FUNCTION_BLOCK ConveyorCTLMultiCast (* Basic Function Block Type *)
  (* Standard: 61499-2 *)
  (* Version 0.2, 2003-12-04, JHC, Rockwell Automation, Renamed for better indexing. *)
  (* Version 0.1, 2002-11-05, JHC, Rockwell Automation, Corrected missing ST element in Algorithm REQ. *)
  (* Version 0.0, 2000-05-30, JHC, Rockwell Automation *)
  (* Compiler header: package fb.rt.cs725; *)
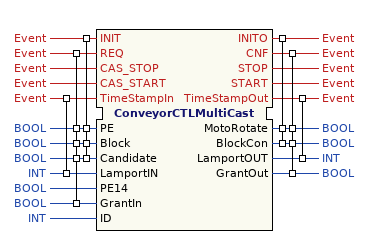
  EVENT_INPUT
    INIT WITH PE, Block, Candidate; (* Initialization Request *)
    REQ WITH PE, Block, Candidate, GrantIn; (* Normal Execution Request *)
    CAS_STOP;
    CAS_START;
    TimeStampIn WITH LamportIN;
  END_EVENT
  EVENT_OUTPUT
    INITO WITH MotoRotate, BlockCon; (* Initialization Confirm *)
    CNF WITH MotoRotate, BlockCon, GrantOut; (* Execution Confirmation *)
    STOP;
    START;
    TimeStampOut WITH LamportOUT;
  END_EVENT
  VAR_INPUT
    PE : BOOL; (* Input event qualifier *)
    Block : BOOL;
    Candidate : BOOL;
    LamportIN : INT;
    PE14 : BOOL;
    GrantIn : BOOL;
    ID : INT;
  END_VAR
  VAR_OUTPUT
    MotoRotate : BOOL; (* Output event qualifier *)
    BlockCon : BOOL;
    LamportOUT : INT;
    GrantOut : BOOL;
  END_VAR
  VAR
    lastPE : BOOL := 1;
    lastBlock : BOOL := 0;
    lamportClock : INT;
  END_VAR
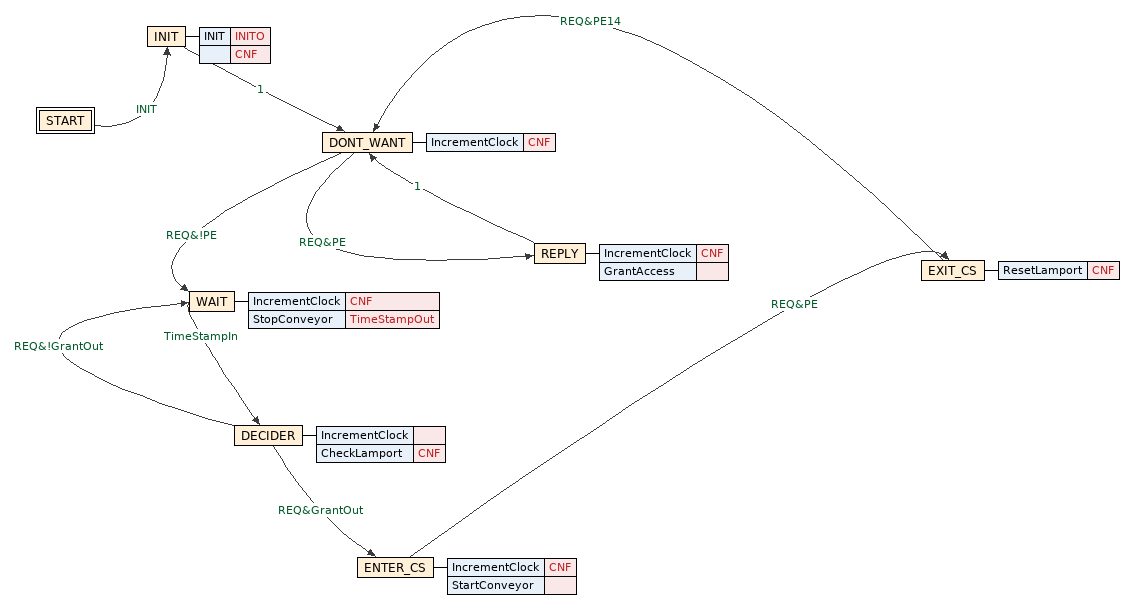
  EC_STATES
    START; (* Initial State *)
    INIT : INIT -> INITO, -> CNF; (* Initialization *)
    WAIT : IncrementClock -> CNF, StopConveyor -> TimeStampOut;
    DONT_WANT : IncrementClock -> CNF;
    REPLY : IncrementClock -> CNF, GrantAccess;
    DECIDER : IncrementClock, CheckLamport -> CNF;
    ENTER_CS : IncrementClock -> CNF, StartConveyor;
    EXIT_CS : ResetLamport -> CNF;
  END_STATES
  EC_TRANSITIONS
    START TO INIT := INIT;
    INIT TO DONT_WANT := 1;
    DONT_WANT TO WAIT := REQ&!PE;
    DONT_WANT TO REPLY := REQ&PE;
    REPLY TO DONT_WANT := 1;
    WAIT TO DECIDER := TimeStampIn;
    DECIDER TO WAIT := REQ&!GrantOut;
    DECIDER TO ENTER_CS := REQ&GrantOut;
    ENTER_CS TO EXIT_CS := REQ&PE;
    EXIT_CS TO DONT_WANT := REQ&PE14;
  END_TRANSITIONS
  ALGORITHM INIT IN ST: (* Initialization algorithm *)
MotoRotate := TRUE;
Block := FALSE;
lamportClock := 0;
GrantOut := FALSE;

System.out.println(this + " " + MotoRotate);
System.out.println(MotoRotate);
  END_ALGORITHM
  ALGORITHM REQ IN ST: (* Normally executed algorithm *)
System.out.println(this +  " -> Candidate" + Candidate);
IF Candidate THEN
IF lastPE !:= PE THEN
IF NOT PE THEN
BlockCon:= TRUE;
System.out.println("BlockCon = true");
ELSE
BlockCon:=FALSE;
System.out.println("BlockCon = false");
END_IF
lastPE := PE;
END_IF
IF lastBlock !:= Block THEN
IF Block THEN
STOP.serviceEvent(this);
MotoRotate := FALSE;
System.out.println("Cas Stop");
ELSE
START.serviceEvent(this);
MotoRotate := TRUE;
System.out.println("Cas Start");
END_IF
lastBlock := Block;
END_IF
END_IF
  END_ALGORITHM
  ALGORITHM START IN ST:
MotoRotate:=TRUE;
System.out.println(this + " Start " + MotoRotate);

System.out.println("Start " + MotoRotate);
  END_ALGORITHM
  ALGORITHM STOP IN ST:
MotoRotate := FALSE;
System.out.println(this + " Stop " + MotoRotate);

System.out.println("Stop " + MotoRotate);
  END_ALGORITHM
  ALGORITHM CheckLamport IN Java:
if(LamportIN.value < lamportClock.value){
GrantOut.value = true;
System.out.println(ID.value + " Own LamportClock is smaller!");
}else if(LamportIN.value > lamportClock.value){
GrantOut.value = false;
System.out.println((ID.value + " Lamport IN is smaller!");
}
  END_ALGORITHM
  ALGORITHM IncrementClock IN Java:
lamportClock.value++;
  END_ALGORITHM
  ALGORITHM GrantAccess IN Java:
GrantOut.value = true;
  END_ALGORITHM
  ALGORITHM StopConveyor IN Java:
GrantOut.value = false;
BlockCon.value = true;
System.out.println(ID.value + " Wait Multicast!");
MotoRotate.value = false;
  END_ALGORITHM
  ALGORITHM StartConveyor IN Java:
BlockCon.value = false;
MotoRotate.value = true;
//System.out.println(ID.value +"Start Conveyer");
  END_ALGORITHM
  ALGORITHM ResetLamport IN Java:
lamportClock.value = 0;
  END_ALGORITHM
END_FUNCTION_BLOCK
